// LS Electric XG5000 project: 71회예상1_1
// PLC NewPLC
// module base 0 slot 0: 입출력 모듈:XBC-DR20S (DC 24V 입력 12점, 릴레이 출력 8점)

PROGRAM NewProgram (task: 스캔 프로그램)

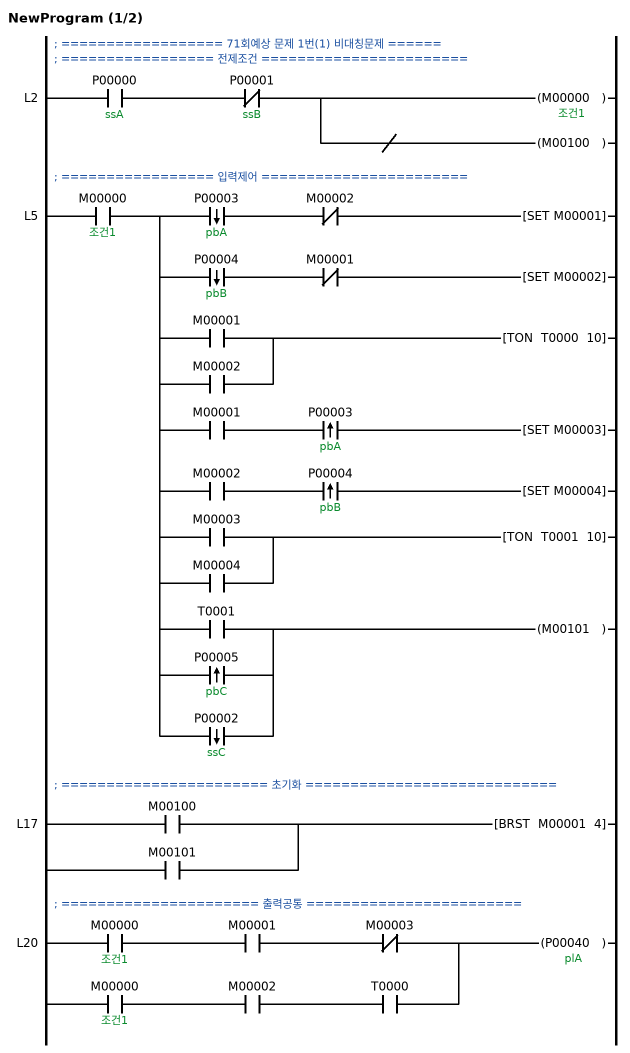
// ================== 71회예상 문제 1번(1) 비대칭문제 ======
// ================= 전제조건 =======================
; L2
LOAD      P00000	// ssA
AND NOT   P00001	// ssB
OUT       M00000	// 조건1
NOT
OUT       M00100
// ================= 입력제어 =======================
; L5
LOAD      M00000	// 조건1
MPUSH
ANDN      P00003	// pbA
AND NOT   M00002
SET       M00001
MLOAD
ANDN      P00004	// pbB
AND NOT   M00001
SET       M00002
MLOAD
LOAD      M00001
OR        M00002
AND LOAD
TON       T0000 10
MLOAD
AND       M00001
ANDP      P00003	// pbA
SET       M00003
MLOAD
AND       M00002
ANDP      P00004	// pbB
SET       M00004
MLOAD
LOAD      M00003
OR        M00004
AND LOAD
TON       T0001 10
MPOP
LOAD      T0001
ORP       P00005	// pbC
ORN       P00002	// ssC
AND LOAD
OUT       M00101
// ======================= 초기화 ============================
; L17
LOAD      M00100
OR        M00101
BRST      M00001 4
// ====================== 출력공통 ========================
; L20
LOAD      M00000	// 조건1
AND       M00001
AND NOT   M00003
LOAD      M00000	// 조건1
AND       M00002
AND       T0000
OR LOAD
OUT       P00040	// plA

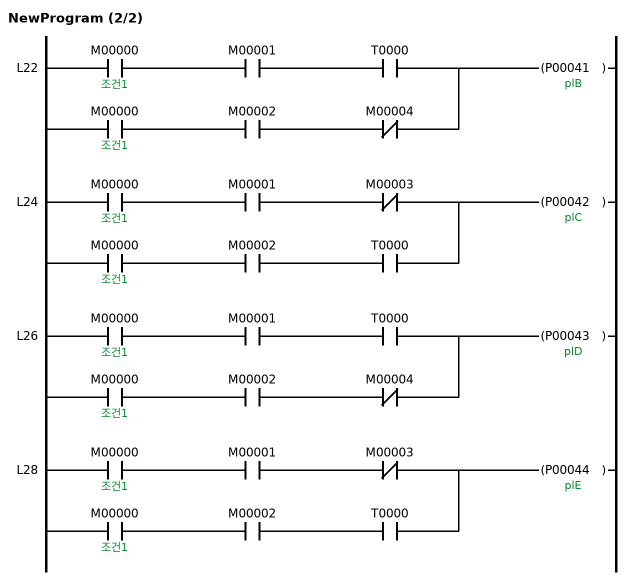
; L22
LOAD      M00000	// 조건1
AND       M00001
AND       T0000
LOAD      M00000	// 조건1
AND       M00002
AND NOT   M00004
OR LOAD
OUT       P00041	// plB
; L24
LOAD      M00000	// 조건1
AND       M00001
AND NOT   M00003
LOAD      M00000	// 조건1
AND       M00002
AND       T0000
OR LOAD
OUT       P00042	// plC
; L26
LOAD      M00000	// 조건1
AND       M00001
AND       T0000
LOAD      M00000	// 조건1
AND       M00002
AND NOT   M00004
OR LOAD
OUT       P00043	// plD
; L28
LOAD      M00000	// 조건1
AND       M00001
AND NOT   M00003
LOAD      M00000	// 조건1
AND       M00002
AND       T0000
OR LOAD
OUT       P00044	// plE